// TIA Portal V18 export
FUNCTION "TEMPLATE--v1.0--00_Only for Commissioning" : Void   // FC1, F_LAD
{ S7_Optimized_Access := 'TRUE' }
// Management of bypass to use during commissioning
BEGIN

REGION Network 1: n0003-mc1-k3201_SN10
   // One network per node
   // TRUE if the node is not ready to be used
   // FALSE if the node is ready
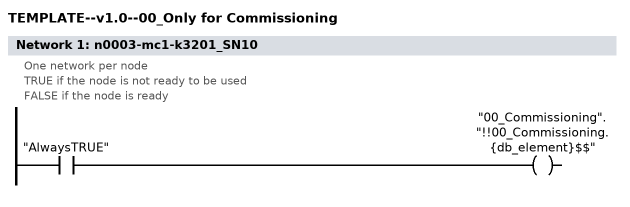
   RUNG wire#powerrail
      Contact( "AlwaysTRUE" )
      Coil( "00_Commissioning"."!!00_Commissioning.{db_element}$$" )
   END_RUNG
   // the same network as SCL:
   "00_Commissioning"."!!00_Commissioning.{db_element}$$" := "AlwaysTRUE";
END_REGION
END_FUNCTION
